Staubli VAL3: printStr.pgx

public program printStr(string& x_sInput[])
  local num l_nElement
  local num l_nLength
begin

  l_nLength = size(x_sInput)

  for l_nElement = 0 to l_nLength-1
    ? x_sInput[l_nElement]
  endFor

end
